FUNCTION_BLOCK ST001_ProcessDataStorage EXTENDS TcoData.TcoDataExchange
VAR
	_data : 
END_VAR

END_FUNCTION_BLOCK

(* stored: Version 1.1.0.1, ProductVersion 3.1.4024.9
   POU ST001_ProcessDataStorage: Id {37e7eeae-cd25-0b59-3f07-4f9672bf8a09}, SpecialFunc None *)
